{attribute addProperty BoxType "EK1122-0000-0018"}
{attribute addProperty Id "Beckhoff_EM3xxxsub_EK1100EK1100_179A0949162"}
{attribute addProperty CRC "883041293"}
{attribute addProperty SizeInBites "16"}
{attribute addProperty SizeInBytes "2"}
TYPE Beckhoff_EM3xxxEK1122_34A2240D EXTENDS EK1122_179A0949 :
STRUCT
	{attribute addProperty Name "Beckhoff_EM3xxxsub_EK1100"}
	Beckhoff_EM3xxxsub_EK1100 : EK1100_179A0949;
END_STRUCT
END_TYPE

(* stored: Version 1.2.0.0, ProductVersion 3.1.4024.9
   DUT Beckhoff_EM3xxxEK1122_34A2240D: Id {ac97cb7c-05c8-43b3-aafc-57044280b270} *)
